// TIA Portal V20 export
VAR_GLOBAL   // PLC tag table "Unit_type"
END_VAR
VAR_GLOBAL CONSTANT   // user constants
   Warehouse1 : Int := 1;
   Warehouse2 : Int := 2;
   Warehouse3 : Int := 3;
   Warehouse4 : Int := 4;
   ShelfGripperPos : Int := 20;
   MC1 : Int := 11;
   MC2 : Int := 12;
   MC3 : Int := 13;
   WarehousePallet : Int := 100;
END_VAR
